PROGRAM TankControl
VAR
	MainState	:	INT;
	FillModeDelay		:	TON;
	DrainModeDelay		:	TON;
END_VAR

FillModeDelay(IN := Pump.LSwitch, PT := T#10S, Q=>,ET=>);
DrainModeDelay(IN := Pump.HSwitch, PT := T#10S, Q=>,ET=>);

IF Pump.LSwitch AND Pump.HSwitch = FALSE THEN
	
	Pump.Pump	:=	FillModeDelay.Q;
	Pump.Valve	:=	FALSE;
	
END_IF

IF Pump.HSwitch AND Pump.LSwitch = FALSE THEN
	
	Pump.Pump	:=	FALSE;
	Pump.Valve	:=	DrainModeDelay.Q;
	
END_IF

END_PROGRAM

(* stored: Version 1.1.0.1, ProductVersion 3.1.4024.9
   POU TankControl: Id {09533a9a-20d9-4d3d-858c-762221111daf}, SpecialFunc None *)
